FUNCTION_BLOCK FB_Machine

VAR_INPUT
	iLogger2 : I_Logger;
END_VAR
VAR
	iLogger : I_Logger;
	
END_VAR

METHOD FB_init : BOOL
VAR_INPUT
	bInitRetains : BOOL; // if TRUE, the retain variables are initialized (warm start / cold start)
	bInCopyCode : BOOL;  // if TRUE, the instance afterwards gets moved into the copy code (online change)
	_iLogger : I_Logger;
END_VAR
iLogger := _iLogger;
END_METHOD

METHOD M_Run : BOOL
VAR_INPUT
	sMessage : STRING(255);
END_VAR

IF iLogger2 <> 0 THEN
	iLogger2.M_Log(sMessage);
END_IF
END_METHOD

END_FUNCTION_BLOCK

(* stored: Version 1.1.0.1, ProductVersion 3.1.4024.16
   POU FB_Machine: Id {33cf73c4-3194-40ea-bb34-68f0dd01cccf}, SpecialFunc None
   Method FB_init: Id {1e42ecf0-b32b-4a14-95c5-0c24950b83c8}
   Method M_Run: Id {092b64db-e74a-4889-9aa3-98d4194dbd68} *)
